// TIA Portal project "Project1" (V18)

(* hardware
DEVICE "S7-1200 station_1"  S7-1200 Station
   slot 0: "Rack_0"  S7-1200 Rack  Rack  V1.0
   slot 1: "PLC_1"  CPU 1214C DC/DC/Rly  6ES7 214-1HG31-0XB0  V3.0
*)

// ===== PLC "PLC_1"  CPU 1214C DC/DC/Rly =====

VAR_GLOBAL   // PLC tag table "Default tag table"
   "iFingers" AT %MW0 : Int;
   "xMainBelt" AT %Q0.0 : Bool;
   "xSorter1_Turn" AT %Q0.3 : Bool;
   "xSorter1_Turn2" AT %Q0.5 : Bool;
   "xSorter1_Turn3" AT %Q0.7 : Bool;
   "xExitConveyor" AT %Q0.2 : Bool;
   "xSorter1_Belt" AT %Q0.4 : Bool;
   "xSorter2_Belt" AT %Q0.6 : Bool;
   "xSorter3_Belt" AT %Q1.0 : Bool;
END_VAR

DATA_BLOCK "DB_FingerCount"   // DB1
{ S7_Optimized_Access := 'FALSE' }
VERSION : 0.1
   VAR
      FingerCount : Int;
   END_VAR
BEGIN
END_DATA_BLOCK

ORGANIZATION_BLOCK "Main"   // OB1, LAD, ProgramCycle
TITLE = "Main Program Sweep (Cycle)"
{ S7_Optimized_Access := 'TRUE' }
VERSION : 0.1
BEGIN

REGION Network 2 (SCL)
   // ============================================================
   // OB1 - Main
   // Sterowanie sorterem na podstawie liczby palców z kamery
   // FingerCount pochodzi z DB1 zapisywanego przez Node-RED
   // ============================================================

   "iFingers" := "DB_FingerCount".FingerCount;

   // Taśma główna i wyjściowa zawsze jadą (oprócz 4-5 palców)
   "xMainBelt" := ("iFingers" >= 0) AND ("iFingers" <= 3);
   "xExitConveyor" := TRUE;

   // Reset sorterów
   "xSorter1_Turn" := FALSE;
   "xSorter1_Turn2" := FALSE;
   "xSorter1_Turn3" := FALSE;
   "xSorter1_Belt" := FALSE;
   "xSorter2_Belt" := FALSE;
   "xSorter3_Belt" := FALSE;

   CASE "iFingers" OF
       0:
           ;
       1:
           "xSorter1_Turn" := TRUE;
           "xSorter1_Belt" := TRUE;
       2:
           "xSorter1_Turn2" := TRUE;
           "xSorter2_Belt" := TRUE;
       3:
           "xSorter1_Turn3" := TRUE;
           "xSorter3_Belt" := TRUE;
       4, 5:
           "xMainBelt" := FALSE;
           "xExitConveyor" := FALSE;
   END_CASE;
END_REGION
END_ORGANIZATION_BLOCK